{attribute 'qualified_only'}
{attribute 'global_init_slot' := '40510'}
VAR_GLOBAL
//elektrozawor siłownika 1
	fbElektrozaworC1						: FB_Elektrozawor_5na2_2Cewki;
//elektrozawor siłownika 2
	fbElektrozaworC2						: FB_Elektrozawor_5na2_2Cewki;
//elektrozawory przesuwacza
	fbElektrozaworPW_Z						: FB_Elektrozawor_5na2_2Cewki;
	fbElektrozaworPW_N						: FB_Elektrozawor_5na2_2Cewki;
END_VAR

(* stored: Version 1.1.0.1, ProductVersion 3.1.4024.11
   GVL GVL_Wyjscia_IO: Id {5939d848-3004-495f-b187-c7f07b9f676e} *)
